(* IEC 61131-3 sources: plc_generation_empirical_study/datasets/task_bank_c06_bounded_runtime_v0_3/tasks/C06_U16_lean_composite, 2 files *)

(* ---- interface.st ---- *)
FUNCTION_BLOCK C06_U16_lean_composite
VAR_INPUT
    A_AddItem : BOOL;
    A_RemoveItem : BOOL;
    A_Reset : BOOL;
    A_Capacity : INT;
    B_Info : BOOL;
    B_Warning : BOOL;
    B_Trip : BOOL;
    B_Emergency : BOOL;
    B_Suppress : BOOL;
    SubsystemBEnable : BOOL;
    CrossReset : BOOL;
END_VAR
VAR_OUTPUT
    A_Count : INT;
    A_Empty : BOOL;
    A_Full : BOOL;
    A_Conflict : BOOL;
    B_Active : BOOL;
    B_Level : INT;
    CrossReady : BOOL;
    CrossBlocked : BOOL;
END_VAR
END_FUNCTION_BLOCK

(* ---- reference.st ---- *)
FUNCTION_BLOCK C06_U16_lean_composite
VAR_INPUT
    A_AddItem : BOOL;
    A_RemoveItem : BOOL;
    A_Reset : BOOL;
    A_Capacity : INT;
    B_Info : BOOL;
    B_Warning : BOOL;
    B_Trip : BOOL;
    B_Emergency : BOOL;
    B_Suppress : BOOL;
    SubsystemBEnable : BOOL;
    CrossReset : BOOL;
END_VAR
VAR_OUTPUT
    A_Count : INT;
    A_Empty : BOOL;
    A_Full : BOOL;
    A_Conflict : BOOL;
    B_Active : BOOL;
    B_Level : INT;
    CrossReady : BOOL;
    CrossBlocked : BOOL;
END_VAR
VAR
    A_PrevAdd : BOOL := FALSE;
    A_PrevRemove : BOOL := FALSE;
END_VAR

A_Conflict := FALSE;
IF A_Reset THEN
    A_Count := 0;
ELSIF A_AddItem AND (NOT A_PrevAdd) AND A_RemoveItem AND (NOT A_PrevRemove) THEN
    A_Conflict := TRUE;
ELSIF A_AddItem AND (NOT A_PrevAdd) AND (A_Count < A_Capacity) THEN
    A_Count := A_Count + 1;
ELSIF A_RemoveItem AND (NOT A_PrevRemove) AND (A_Count > 0) THEN
    A_Count := A_Count - 1;
END_IF;
A_Empty := A_Count = 0;
A_Full := A_Count >= A_Capacity;
A_PrevAdd := A_AddItem;
A_PrevRemove := A_RemoveItem;

IF CrossReset THEN
    CrossReady := FALSE;
ELSIF A_Empty THEN
    CrossReady := TRUE;
END_IF;
CrossBlocked := SubsystemBEnable AND (NOT CrossReady);

IF SubsystemBEnable AND CrossReady THEN
    IF B_Emergency THEN
        B_Level := 4;
        B_Active := TRUE;
    ELSIF B_Suppress THEN
        B_Level := 0;
        B_Active := FALSE;
    ELSIF B_Trip THEN
        B_Level := 3;
        B_Active := TRUE;
    ELSIF B_Warning THEN
        B_Level := 2;
        B_Active := TRUE;
    ELSIF B_Info THEN
        B_Level := 1;
        B_Active := TRUE;
    ELSE
        B_Level := 0;
        B_Active := FALSE;
    END_IF;
ELSE
    B_Active := FALSE;
    B_Level := 0;
END_IF;

END_FUNCTION_BLOCK
